// TIA Portal V20 export
DATA_BLOCK "HmiInterface"   // DB82
// stored: Access Published, MemoryReserve 100, Namespace Unit1.Em8
   VAR
      em : "LAF_typeEmInterface";
      cm : "Unit1.Em8.typeCmHmiInterface";
      hipotThickness : "LER_typeSequenceInterface";
      GRnR_hipotThickness { S7_SetPoint := 'True'} : "LER_typeSequenceInterface";
      cmHipotThicknessSafetyPin : "LBC_typeDigitalSignalInterface";
      cmHipotThicknessJRDetect : "LBC_typeDigitalSignalInterface";
   END_VAR
   VAR RETAIN
      cmThicknessAxisZ : "LBC_typeAxis64PosInterface";
   END_VAR
   VAR
      cmHipotThicknessStageLiftFrontUpDown : "LBC_typeTwoWayActuatorInterface";
      cmHipotThicknessStageLiftRearUpDown : "LBC_typeTwoWayActuatorInterface";
      cmHipotTabContactorBwdFwd : "LBC_typeTwoWayActuatorInterface";
      cmHipotTabContactorLeftOpenClose : "LBC_typeTwoWayActuatorInterface";
      cmHipotTabContactorRightOpenClose : "LBC_typeTwoWayActuatorInterface";
      cmHipotThicknessStageLiftAllUpDown : "LBC_typeTwoWayActuatorInterface";
      cmHipotThicknessServoPress : "LER_typeServoPressInterface";
      cmThicknessControl : "LER_typeThicknessInterface";
      cmHipotControl : "LER_typeHipotInterface";
      cmHipotThicknessServoPressHistory : "LER_typeServoPressHistory";
      cmHipotHistory : "LER_typeHipotHistory";
      cmThicknessHistory : "LER_typeThicknessHistory";
      "cmThicknessHistory_r&r" : "LER_typeThicknessHistory_R&R";
      gaugeRnR : "Unit1.Em8.typeGaugeRnRHmiInterface";
      HipotRepeat : "Unit1.Em8.typeHipotRepeatHmiInterface";
      HipotRepeatUnuse : Bool;
      intCondition : "Unit1.Em8.typeIntConditionHmiInterface";
   END_VAR
BEGIN
   cmHipotControl.configuration.port := 1054;
END_DATA_BLOCK
